FUNCTION_BLOCK FB_MalzemeSecme
VAR_INPUT
	nValue: INT;
END_VAR
VAR_OUTPUT
	nStateOut: INT;
	sMsg: STRING;
END_VAR
VAR
END_VAR



IF nValue >= 0 AND nValue <=40 THEN
	
	sMsg := 'Malzeme Kısa Boyutlu.';
	
	nStateOut := 32;
	
ELSIF nValue >40 AND nValue <= 70 THEN

	sMsg := 'Malzeme Orta Boyutlu.';
	nStateOut := 34;
	
ELSIF nValue > 70 AND nValue <=100 THEN
		
	sMsg := 'Malzeme Uzun Boyutlu.';
	nStateOut := 36;	
	
END_IF

END_FUNCTION_BLOCK

(* stored: Version 1.1.0.1, ProductVersion 3.1.4024.4
   POU FB_MalzemeSecme: Id {8e663e0a-af29-4c9f-901d-da0bace0c49c}, SpecialFunc None *)
